FUNCTION_BLOCK Test_ReadBySymbolName_KeepingHandle EXTENDS TUnitTestBase
VAR
    AdsReadBySymbolName : TAdsReadBySymbolName;
    ValueToRead : INT;
    ReadResult  : INT;
    ScanCount : DINT;
    State: INT;
END_VAR

CASE State OF
    0:
        ValueToRead := 1234;
        ReadResult := 0;
        ScanCount := 0;
    
        AdsReadBySymbolName.Execute(
            AmsNetId:= '', 
            Port:= 851, 
            SymbolName:= 'PB_TestRunner.Test_ReadBySymbolName_KeepingHandle.ValueToRead', 
            ReadDataAddress:= ADR(ReadResult), 
            ReadDataLength:= SIZEOF(ReadResult), 
            KeepSymbolHandle:= TRUE);

        State := 10;
        
    10:
        ScanCount := ScanCount + 1;
        IF NOT AdsReadBySymbolName.Execution.Busy THEN
            State := 20;    
		END_IF
        
    20:
        Assertion.AssertEquals_INT(
            Expected     := 1234,
            Actual       := ReadResult,
            ObjectName   := _TestName,
            Variablename := 'ReadResult'); 
 
        TestFinished();
        State := 0;
END_CASE

AdsReadBySymbolName();

END_FUNCTION_BLOCK

(* stored: Version 1.1.0.1, ProductVersion 3.1.4024.3
   POU Test_ReadBySymbolName_KeepingHandle: Id {9946ec85-dcda-05bf-0580-cea8be438229}, SpecialFunc None *)
